// TwinCAT 3 PLC project PLC_ProcessControl
// ProgramVersion: 3.1.4026.19
// CompilerDefines: VISU_USEPROPERTYINFO
// libraries:
//   Tc2_Standard, * (Beckhoff Automation GmbH)
//   Tc2_System, * (Beckhoff Automation GmbH)
//   VisuDialogs, * (System)
//   VisuSymbols, 4.5.0.0 (System)
// project tree:
//   DUTs/ stRecipe.TcDUT
//   / GlobalTextList.TcGTLO, PlcTask.TcTTO, Visualization Manager.TcVMO (not stored)
//   GVLs/ GVL_Process.TcGVL
//   POUs/ MAIN.TcPOU
//   VISUs/ Visualization.TcVIS
// real-time tasks:
//   TASK PlcTask: cycle T#10ms, priority 20, ADS port 350

CONFIGURATION PLC_ProcessControl
    RESOURCE PLC ON TwinCAT3
        TASK PlcTask(INTERVAL := T#10ms, PRIORITY := 20);
        PROGRAM MAIN WITH PlcTask : MAIN;
    END_RESOURCE
END_CONFIGURATION

// ---- DUTs/stRecipe.TcDUT
TYPE stRecipe :
STRUCT
	sProductName : STRING(50);
	fTargetFill_ml : REAL;
	fTargetTemp_Celsius : REAL;
	tMixingDuration : TIME;
END_STRUCT
END_TYPE

// ---- GVLs/GVL_Process.TcGVL
VAR_GLOBAL
    // --- Recipe Management ---
    astRecipes      : ARRAY[1..3] OF stRecipe;
    stCurrentRecipe : stRecipe;
    nSelectedRecipe : INT := 1;     // 1=Cola, 2=Juice
    
    // --- HMI Visual Feedback & UI ---
    bColaActive     : BOOL;         
    bJuiceActive    : BOOL;         
    sStatusMessage  : STRING(50);   
    sCurrentProduct : STRING(50);   // NEW: Currently running product name
    
    // --- Production Stats (OEE - Counters) ---
    nTotalBottles   : INT := 0;     // Total bottles
    nColaCount      : INT := 0;     // NEW: Cola counter
    nJuiceCount     : INT := 0;     // NEW: Juice counter
    
    // --- Process Values (Sensors) ---
    fCurrentTemp    : REAL;
    fCurrentLevel   : REAL;
    
    // --- Control Signals (Buttons & Safety) ---
    bStartProcess   : BOOL;         // Acts as Continuous Run Flag
    bEmergencyStop  : BOOL;
    
    // --- Actuators (Outputs) ---
    bInletValve     : BOOL;
    bOutletValve    : BOOL;
    bHeater         : BOOL;
    bMixerMotor     : BOOL;
	
// --- Predictive Maintenance 
    nValveCycleCount       : INT := 0;     
    nRandomThreshold       : INT := 5;    
    bMaintenanceAlarm      : BOOL;   
END_VAR

// ---- POUs/MAIN.TcPOU
PROGRAM MAIN
VAR
    // --- The Brain: State Machine ---
    // YENİ EKLENDİ: STATE_MAINTENANCE
    eState : (STATE_IDLE, STATE_INIT, STATE_FILLING, STATE_HEATING, STATE_MIXING, STATE_BOTTLING, STATE_COMPLETE, STATE_MAINTENANCE, STATE_ERROR) := STATE_IDLE;
    
    // --- Timers & Triggers ---
    fbTimerMixing   : TON; 
    rtInletValve    : R_TRIG;
    
    // --- Simulation Rates ---
    fFillRate       : REAL := 2.5;  
    fHeatRate       : REAL := 0.1;  
    fEmptyRate      : REAL := 2.5;  
END_VAR

// =========================================================
// 0. HMI VISUAL FEEDBACK & STATUS MAP
// =========================================================
GVL_Process.bColaActive  := (GVL_Process.nSelectedRecipe = 1);
GVL_Process.bJuiceActive := (GVL_Process.nSelectedRecipe = 2);


// =========================================================
// 0.5 PREDICTIVE MAINTENANCE 
// =========================================================
rtInletValve(CLK := GVL_Process.bInletValve);

IF rtInletValve.Q THEN
    GVL_Process.nValveCycleCount := GVL_Process.nValveCycleCount + 1;
END_IF


IF GVL_Process.nValveCycleCount >= GVL_Process.nRandomThreshold AND eState <> STATE_MAINTENANCE AND eState <> STATE_ERROR THEN
    GVL_Process.bMaintenanceAlarm := TRUE;
    eState := STATE_MAINTENANCE; 
END_IF


// =========================================================
// 1. SAFETY FIRST: EMERGENCY STOP OVERRIDE
// =========================================================
IF GVL_Process.bEmergencyStop THEN
    eState := STATE_ERROR;
    GVL_Process.bStartProcess := FALSE; // Cancel continuous run on error
END_IF

// =========================================================
// 2. MAIN PROCESS: STATE MACHINE
// =========================================================
CASE eState OF

    STATE_IDLE: 
        GVL_Process.sStatusMessage := 'SYSTEM READY - WAITING FOR START';
        GVL_Process.sCurrentProduct := '-'; // Clear product screen
        
        // Loop starts here and keeps bStartProcess TRUE
        IF GVL_Process.bStartProcess AND NOT GVL_Process.bEmergencyStop THEN
            eState := STATE_INIT;
        END_IF

    STATE_INIT: 
        GVL_Process.sStatusMessage := 'INITIALIZING RECIPE...';
        
        // --- DYNAMIC RECIPE SELECTION ---
        IF GVL_Process.nSelectedRecipe = 1 THEN
            GVL_Process.stCurrentRecipe.sProductName := 'Cola';
            GVL_Process.stCurrentRecipe.fTargetFill_ml := 1000.0;
            GVL_Process.stCurrentRecipe.fTargetTemp_Celsius := 85.0;
            GVL_Process.stCurrentRecipe.tMixingDuration := T#5S;
            GVL_Process.sCurrentProduct := 'COLA'; // HMI Update
            
        ELSIF GVL_Process.nSelectedRecipe = 2 THEN
            GVL_Process.stCurrentRecipe.sProductName := 'Juice';
            GVL_Process.stCurrentRecipe.fTargetFill_ml := 800.0;
            GVL_Process.stCurrentRecipe.fTargetTemp_Celsius := 70.0;
            GVL_Process.stCurrentRecipe.tMixingDuration := T#3S;
            GVL_Process.sCurrentProduct := 'JUICE'; // HMI Update
        END_IF
        
        // Reset outputs for the new bottle
        GVL_Process.bInletValve  := FALSE;
        GVL_Process.bHeater      := FALSE;
        GVL_Process.bMixerMotor  := FALSE;
        GVL_Process.bOutletValve := FALSE;
        GVL_Process.fCurrentLevel := 0.0;
        GVL_Process.fCurrentTemp  := 20.0; 
        
        eState := STATE_FILLING;

    STATE_FILLING: 
        GVL_Process.sStatusMessage := 'FILLING TANK...';
        GVL_Process.bInletValve := TRUE;
        
        GVL_Process.fCurrentLevel := GVL_Process.fCurrentLevel + fFillRate;
        
        IF GVL_Process.fCurrentLevel >= GVL_Process.stCurrentRecipe.fTargetFill_ml THEN
            GVL_Process.fCurrentLevel := GVL_Process.stCurrentRecipe.fTargetFill_ml; 
            GVL_Process.bInletValve := FALSE; 
            eState := STATE_HEATING;
        END_IF

    STATE_HEATING: 
        GVL_Process.sStatusMessage := 'HEATING PRODUCT...';
        GVL_Process.bHeater := TRUE;
        
        GVL_Process.fCurrentTemp := GVL_Process.fCurrentTemp + fHeatRate;
        
        IF GVL_Process.fCurrentTemp >= GVL_Process.stCurrentRecipe.fTargetTemp_Celsius THEN
            GVL_Process.fCurrentTemp := GVL_Process.stCurrentRecipe.fTargetTemp_Celsius; 
            GVL_Process.bHeater := FALSE; 
            eState := STATE_MIXING;
        END_IF

    STATE_MIXING: 
        GVL_Process.sStatusMessage := 'MIXING INGREDIENTS...';
        GVL_Process.bMixerMotor := TRUE;
        fbTimerMixing(IN := TRUE, PT := GVL_Process.stCurrentRecipe.tMixingDuration);
        
        IF fbTimerMixing.Q THEN 
            GVL_Process.bMixerMotor := FALSE;
            fbTimerMixing(IN := FALSE); 
            eState := STATE_BOTTLING;
        END_IF

    STATE_BOTTLING: 
        GVL_Process.sStatusMessage := 'BOTTLING PRODUCT...';
        GVL_Process.bOutletValve := TRUE;
        
        GVL_Process.fCurrentLevel := GVL_Process.fCurrentLevel - fEmptyRate;
        
        IF GVL_Process.fCurrentLevel <= 0.0 THEN
            GVL_Process.fCurrentLevel := 0.0; 
            GVL_Process.bOutletValve := FALSE;
            eState := STATE_COMPLETE;
        END_IF

    STATE_COMPLETE: 
        GVL_Process.sStatusMessage := 'BATCH COMPLETE!';
        GVL_Process.nTotalBottles := GVL_Process.nTotalBottles + 1; 
        
        // --- SEPARATE COUNTERS ---
        IF GVL_Process.nSelectedRecipe = 1 THEN
            GVL_Process.nColaCount := GVL_Process.nColaCount + 1;
        ELSIF GVL_Process.nSelectedRecipe = 2 THEN
            GVL_Process.nJuiceCount := GVL_Process.nJuiceCount + 1;
        END_IF
        
        // --- CONTINUOUS LOOP LOGIC ---
        IF GVL_Process.bStartProcess THEN
            eState := STATE_INIT; // Start logic is still ON, jump to next bottle!
        ELSE
            eState := STATE_IDLE; // Start was turned OFF, go to sleep.
        END_IF

STATE_MAINTENANCE: 
        GVL_Process.sStatusMessage := 'CRITICAL: HIGH VIBRATION & TEMP! MAINTENANCE REQUIRED!';
        
        // Sistemi güvenliğe al ve durdur
        GVL_Process.bInletValve  := FALSE;
        GVL_Process.bHeater      := FALSE;
        GVL_Process.bMixerMotor  := FALSE;
        GVL_Process.bOutletValve := FALSE;
        fbTimerMixing(IN := FALSE);
        GVL_Process.bStartProcess := FALSE; // Sürekli üretimi iptal et!
        
        
        IF NOT GVL_Process.bMaintenanceAlarm THEN
            GVL_Process.nRandomThreshold := 5;
            
            GVL_Process.nValveCycleCount := 0;
            eState := STATE_IDLE;
        END_IF

    STATE_ERROR: 
        GVL_Process.sStatusMessage := 'SYSTEM LOCKED - EMERGENCY STOP!';
        GVL_Process.bInletValve  := FALSE;
        GVL_Process.bHeater      := FALSE;
        GVL_Process.bMixerMotor  := FALSE;
        GVL_Process.bOutletValve := FALSE;
        fbTimerMixing(IN := FALSE);
        
        // E-Stop reset & Start
        IF NOT GVL_Process.bEmergencyStop AND GVL_Process.bStartProcess THEN
             GVL_Process.bStartProcess := FALSE;
             eState := STATE_IDLE;
        END_IF

END_CASE

END_PROGRAM

// ---- GlobalTextList.TcGTLO
TEXTLIST GlobalTextList
  582 = 'Cola'
  536 = 'Cola Produced: %i'
  854 = 'Cola Produced: %s'
  755 = 'Emergency Stop'
  712 = 'HEATING'
  294 = 'Juice'
  162 = 'Juice Produced: %i'
  554 = 'MIXER'
  699 = 'Now Producing: %s'
  891 = 'Nsad'
  505 = 'Orange Saft'
  361 = 'Start Process'
  745 = 'Status:'
  971 = 'Status: %s'
  803 = 'Stop Process'
  362 = 'System is locked! Emergency!!!'
  867 = 'SYSTEM SHUT DOWN HIGH HEAT AND VIBRATION DETECTED!'
  461 = 'System shut down!\n\nHigh heat and vibration detected!'
  940 = 'System shut down!\n\nHigh heat and vibration detected! Click to perform maintenance'
  716 = 'System shut down!\n\nHigh heat and vibration detected! Click to perform maintenance!'
  627 = 'System shut down!\n\nHigh heat and vibration detected!Click to perform maintenance!'
  189 = 'System shut down!\n\n\nHigh heat and vibration detected!\n\nClick to perform maintenance!'
  296 = 'System shut down!\n\n\n\nHigh heat and vibration detected!\n\nClick to perform maintenance!'
  549 = 'System shut down! \n\nHigh heat and vibration detected!\n\nClick to perform maintenance!'
  260 = 'SYSTEM SHUT DOWN: HIGH HEAT AND VIBRATION DETECTED!'
  859 = 'TANK'
  101 = 'TANK LEVEL'
  801 = 'Tank Level'
  424 = 'Temperature'
  382 = 'Total Bottles Produced: %i'
  402 = 'VALF'
  280 = 'Valve Cycles: %i'
  567 = 'Valve Cycles: %i / %i'
END_TEXTLIST

// ---- VISUs/Visualization.TcVIS
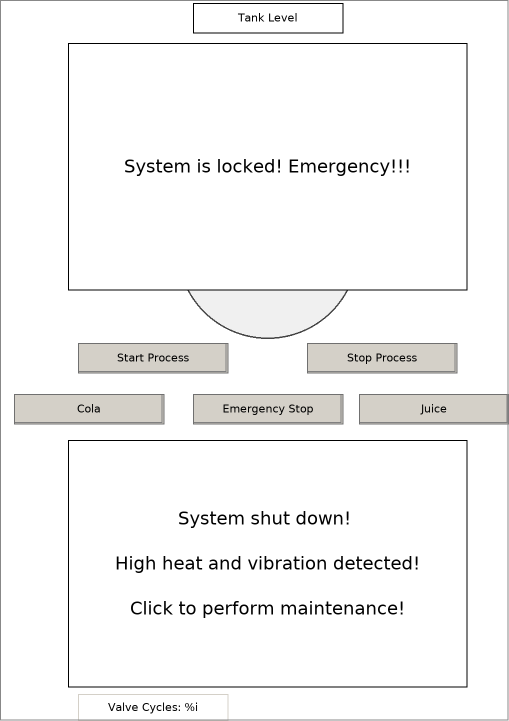
VISUALIZATION Visualization  // 509x721
    BarDisplayImage (119,43 300x50), value: GVL_Process.fCurrentLevel, style: BarDisplayImage-Gray, scale format: %.1f, scale 0..1000
    Meter360 (177,150 181x196), value: GVL_Process.fCurrentTemp, style: Meter-Meter360-Gray, scale format: %.1f, scale 0..100
    Rectangle (193,3 150x30), "Tank Level"
    Rectangle (193,103 150x30), "Temperature"
    Button (78,343 150x30), "Start Process"
        OnMouseClick: execute { GVL_Process.bStartProcess := TRUE; }
    Button (193,394 150x30), "Emergency Stop"
        toggle GVL_Process.bEmergencyStop
    Button (14,394 150x30), "Cola"
        tap GVL_Process.bColaActive
        OnMouseClick: execute { GVL_Process.nSelectedRecipe := 1; }
    Button (359,394 150x30), "Juice"
        tap GVL_Process.bJuiceActive
        OnMouseClick: execute { GVL_Process.nSelectedRecipe := 2; }
    Rectangle (102,520 78x18), "VALF"
    Rectangle (233,520 78x18), "HEATING"
    Rectangle (359,520 78x18), "MIXER"
    Lamp1 (110,440 70x70), variable: GVL_Process.bInletValve, style: Lamp-Lamp1-Yellow
    Lamp1 (241,440 70x70), variable: GVL_Process.bHeater, style: Lamp-Lamp1-Yellow
    Lamp1 (359,440 70x70), variable: GVL_Process.bMixerMotor, style: Lamp-Lamp1-Yellow
    Textfield (78,599 150x30), "Total Bottles Produced: %i", text variable: GVL_Process.nTotalBottles
    Rectangle (68,43 399x247), "System is locked! Emergency!!!", invisible if: NOT GVL_Process.bEmergencyStop
    Textfield (78,554 372x28), "Status: %s", text variable: GVL_Process.sStatusMessage
    Button (307,343 150x30), "Stop Process"
        OnMouseClick: execute { GVL_Process.bStartProcess := FALSE; }
    Textfield (279,599 150x30), "Cola Produced: %i", text variable: GVL_Process.nColaCount
    Textfield (78,644 150x30), "Now Producing: %s", text variable: GVL_Process.sCurrentProduct
    Textfield (279,644 150x30), "Juice Produced: %i", text variable: GVL_Process.nJuiceCount
    Textfield (78,694 150x27), "Valve Cycles: %i", text variable: GVL_Process.nValveCycleCount
    Rectangle (68,440 399x247), "System shut down! High heat and vibration detected! Click to perform maintenance!", invisible if: NOT GVL_Process.bMaintenanceAlarm
        OnMouseClick: execute { GVL_Process.bMaintenanceAlarm := FALSE; }
END_VISUALIZATION
